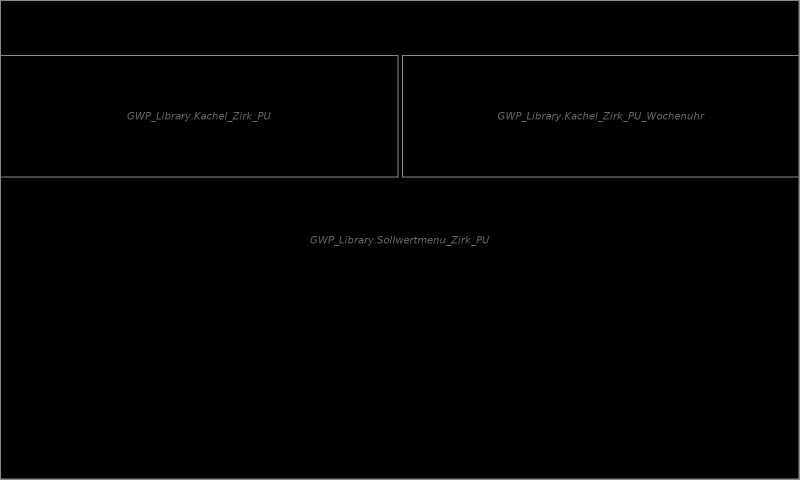
VISUALIZATION Sollwertmenu_Zirk_PU  // 800x480
    Frame (0,0 800x480)
        shows GWP_Library.Sollwertmenu_Zirk_PU(FB_Init_1 := Main.Init_0)
    Frame (0,55 398x122)
        shows GWP_Library.Kachel_Zirk_PU()
        OnMouseClick: change screen: Zirkulationspumpe_Sollwerte
    Frame (402,55 398x122)
        shows GWP_Library.Kachel_Zirk_PU_Wochenuhr()
        OnMouseClick: change screen: Zirkulationspumpe_CLK_W7_Siebentageprogramm
END_VISUALIZATION

(* stored: Version 1.1.0.1, ProductVersion 3.1.4022.6
   Visu Sollwertmenu_Zirk_PU: Id {8bb6e17e-af7d-4b42-adaf-90243c9ec28d} *)
